// TIA Portal V18 export
TYPE "UDT_BoilerOpMode"
// stored: IsFailsafeCompliant false
   STRUCT
      cPreviousOne { S7_SetPoint := 'True'} : Array[1..2] of Byte;
      cActual { S7_SetPoint := 'True'} : Array[1..2] of Byte;   // Поточний/Актуальний режим роботи
      cTarget { S7_SetPoint := 'True'} : Array[1..2] of Byte;   // Вибраний режим роботи, але ще не дійшли до нього
      cPreselectedOpModePLC : Array[1..2] of Byte;   // Вибор режиму роботи з PLC. 0-Вимкенено/1-Boiler1/2-Boiler2/3-B1+B2/4-Auto
      cReserve : Array[1..2] of Byte;
      cPreselectedOpModePanel : Array[1..2] of Byte;   // Вибор режиму роботи з Фізичного перемикача на шафы. 0-Summer/1-Winter/2--Auto
      xBoiler2IndividualPanelSwitch : Bool;
   END_STRUCT;
END_TYPE
